FUNCTION DialogCheckInit : BOOL
VAR_IN_OUT
	stValue : STRING;
	stOutput : STRING;
	bInit : BOOL;
END_VAR
VAR
END_VAR

IF bInit THEN
	stValue := ''; 
	stOutput := '';
	g_XExp := FALSE;
	// g_Format is reset on close, not on init
	bInit := FALSE;
END_IF

END_FUNCTION

(* stored: Version 1.1.0.1, ProductVersion 3.1.4024.2
   POU DialogCheckInit: Id {58a5f58b-ffa1-4982-a209-36f8d1d5471a}, SpecialFunc None *)
